TYPE ST_VirtualHeatCounterDefaultParameters_Storage:
STRUCT
	tTaskCycleTime	: TIME;
	tCtrlCycleTime	: TIME;
	fHeatCapacity : REAL := 4180; //kJ/K
END_STRUCT
END_TYPE

(* stored: Version 1.1.0.1, ProductVersion 3.1.4024.10
   DUT ST_VirtualHeatCounterDefaultParameters_Storage: Id {fd8c7033-668e-4b7c-8f48-c375e60398f8} *)
